Fanuc TP program (LS listing): CLEAR_MSG.LS

/PROG  CLEAR_MSG
/ATTR
OWNER		= MNEDITOR;
COMMENT		= "";
PROG_SIZE	= 232;
CREATE		= DATE 26-08-28  TIME 19:39:30;
MODIFIED	= DATE 26-08-28  TIME 19:40:32;
FILE_NAME	= ;
VERSION		= 0;
LINE_COUNT	= 10;
MEMORY_SIZE	= 564;
PROTECT		= READ_WRITE;
TCD:  STACK_SIZE	= 0,
      TASK_PRIORITY	= 50,
      TIME_SLICE	= 0,
      BUSY_LAMP_OFF	= 0,
      ABORT_REQUEST	= 0,
      PAUSE_REQUEST	= 0;
DEFAULT_GROUP	= 1,*,*,*,*;
CONTROL_CODE	= 00000000 00000000;
/MN
   1:  MESSAGE[ ] ;
   2:  MESSAGE[ ] ;
   3:  MESSAGE[ ] ;
   4:  MESSAGE[ ] ;
   5:  MESSAGE[ ] ;
   6:  MESSAGE[ ] ;
   7:  MESSAGE[ ] ;
   8:  MESSAGE[ ] ;
   9:  MESSAGE[ ] ;
  10:  MESSAGE[ ] ;
/POS
/END
